Fanuc KAREL source: NC0031.KL

-- PROVISIONAL review KL for V1013-1; original PC SHA256 d6147291fd4dc6949de40ecb1147e79c050cf0ada10eea68c805d8dba57ce3dc
-- Incomplete behavior may be omitted. Consult companion uncertainty JSON. Do not deploy.
PROGRAM NC0031
%NOLOCKGROUP
-- UNRESOLVED_LOCAL_POOL 1 cells at code offset 3; source declarations unknown
-- DIRECT_LOCAL_WORD_ACCESS alone does not prove INTEGER, REAL, or BOOLEAN
BEGIN
  -- UNRESOLVED_PC offsets 0-8; opcodes 2B,2C,7B
  -- UNRESOLVED_PC offsets 13-20; opcodes 9D,23
  -- UNRESOLVED_PC offsets 25-42; opcodes 21,40,41,42
  -- UNRESOLVED_PC offsets 47-64; opcodes 21,40,41,42
  -- UNRESOLVED_PC offsets 69-86; opcodes 21,40,41,42
  -- UNRESOLVED_PC offsets 91-108; opcodes 21,40,41,42
  -- UNRESOLVED_PC offsets 113-130; opcodes 21,40,41,42
  -- UNRESOLVED_PC offsets 135-152; opcodes 21,40,41,42
  -- UNRESOLVED_PC offsets 157-174; opcodes 21,40,41,42
  -- UNRESOLVED_PC offsets 179-196; opcodes 21,40,41,42
  -- UNRESOLVED_PC offsets 201-218; opcodes 21,40,41,42
  -- UNRESOLVED_PC offsets 223-240; opcodes 21,40,41,42
  -- UNRESOLVED_PC offsets 245-262; opcodes 21,40,41,42
  -- UNRESOLVED_PC offsets 267-284; opcodes 21,40,41,42
  -- UNRESOLVED_PC offsets 289-306; opcodes 21,40,41,42
  -- UNRESOLVED_PC offsets 311-328; opcodes 21,40,41,42
  -- UNRESOLVED_PC offsets 333-350; opcodes 21,40,41,42
  -- UNRESOLVED_PC offsets 355-372; opcodes 21,40,41,42
  -- UNRESOLVED_PC offsets 377-394; opcodes 21,40,41,42
  -- UNRESOLVED_PC offsets 399-416; opcodes 21,40,41,42
  -- UNRESOLVED_PC offsets 421-438; opcodes 21,40,41,42
  -- UNRESOLVED_PC offsets 443-460; opcodes 21,40,41,42
  -- UNRESOLVED_PC offsets 465-495; opcodes 21,9D,52,23,7A,40,41,42
  -- UNRESOLVED_PC offsets 500-524; opcodes 21,2E,52,23,7A,43
  -- UNRESOLVED_PC offsets 529-547; opcodes 21,2E,52,23
  -- UNRESOLVED_PC offsets 552-568; opcodes 7A,40,41,42
  -- UNRESOLVED_PC offsets 573-597; opcodes 21,2E,52,23,7A,43
  -- UNRESOLVED_PC offsets 602-620; opcodes 21,2E,52,23
  -- UNRESOLVED_PC offsets 625-641; opcodes 7A,40,41,42
  -- UNRESOLVED_PC offsets 646-670; opcodes 21,2E,52,23,7A,43
  -- UNRESOLVED_PC offsets 675-693; opcodes 21,2E,52,23
  -- UNRESOLVED_PC offsets 698-714; opcodes 7A,40,41,42
  -- UNRESOLVED_PC offsets 719-743; opcodes 21,2E,52,23,7A,43
  -- UNRESOLVED_PC offsets 748-766; opcodes 21,2E,52,23
  -- UNRESOLVED_PC offsets 771-787; opcodes 7A,40,41,42
  -- UNRESOLVED_PC offsets 792-816; opcodes 21,2E,52,23,7A,43
  -- UNRESOLVED_PC offsets 821-839; opcodes 21,2E,52,23
  -- UNRESOLVED_PC offsets 844-860; opcodes 7A,40,41,42
  -- UNRESOLVED_PC offsets 865-889; opcodes 21,2E,52,23,7A,43
  -- UNRESOLVED_PC offsets 894-912; opcodes 21,2E,52,23
  -- UNRESOLVED_PC offsets 917-933; opcodes 7A,40,41,42
  -- UNRESOLVED_PC offsets 938-962; opcodes 21,2E,52,23,7A,43
  -- UNRESOLVED_PC offsets 967-985; opcodes 21,2E,52,23
  -- UNRESOLVED_PC offsets 990-1006; opcodes 7A,40,41,42
  -- UNRESOLVED_PC offsets 1011-1035; opcodes 21,2E,52,23,7A,43
  -- UNRESOLVED_PC offsets 1040-1058; opcodes 21,2E,52,23
  -- UNRESOLVED_PC offsets 1063-1079; opcodes 7A,40,41,42
  -- UNRESOLVED_PC offsets 1084-1108; opcodes 21,2E,52,23,7A,43
  -- UNRESOLVED_PC offsets 1113-1131; opcodes 21,2E,52,23
  -- UNRESOLVED_PC offsets 1136-1152; opcodes 7A,40,41,42
  -- UNRESOLVED_PC offsets 1157-1181; opcodes 21,2E,52,23,7A,43
  -- UNRESOLVED_PC offsets 1186-1204; opcodes 21,2E,52,23
  -- UNRESOLVED_PC offsets 1209-1225; opcodes 7A,40,41,42
  -- UNRESOLVED_PC offsets 1230-1254; opcodes 21,2E,52,23,7A,43
  -- UNRESOLVED_PC offsets 1259-1277; opcodes 21,2E,52,23
  -- UNRESOLVED_PC offsets 1282-1298; opcodes 7A,40,41,42
  -- UNRESOLVED_PC offsets 1303-1327; opcodes 21,2E,52,23,7A,43
  -- UNRESOLVED_PC offsets 1332-1350; opcodes 21,2E,52,23
  -- UNRESOLVED_PC offsets 1355-1371; opcodes 7A,40,41,42
  -- UNRESOLVED_PC offsets 1376-1400; opcodes 21,2E,52,23,7A,43
  -- UNRESOLVED_PC offsets 1405-1423; opcodes 21,2E,52,23
  -- UNRESOLVED_PC offsets 1428-1444; opcodes 7A,40,41,42
  -- UNRESOLVED_PC offsets 1449-1473; opcodes 21,2E,52,23,7A,43
  -- UNRESOLVED_PC offsets 1478-1496; opcodes 21,2E,52,23
  -- UNRESOLVED_PC offsets 1501-1517; opcodes 7A,40,41,42
  -- UNRESOLVED_PC offsets 1522-1546; opcodes 21,2E,52,23,7A,43
  -- UNRESOLVED_PC offsets 1551-1569; opcodes 21,2E,52,23
  -- UNRESOLVED_PC offsets 1574-1590; opcodes 7A,40,41,42
  -- UNRESOLVED_PC offsets 1595-1619; opcodes 21,2E,52,23,7A,43
  -- UNRESOLVED_PC offsets 1624-1642; opcodes 21,2E,52,23
  -- UNRESOLVED_PC offsets 1647-1663; opcodes 7A,40,41,42
  -- UNRESOLVED_PC offsets 1668-1692; opcodes 21,2E,52,23,7A,43
  -- UNRESOLVED_PC offsets 1697-1715; opcodes 21,2E,52,23
  -- UNRESOLVED_PC offsets 1720-1736; opcodes 7A,40,41,42
  -- UNRESOLVED_PC offsets 1741-1765; opcodes 21,2E,52,23,7A,43
  -- UNRESOLVED_PC offsets 1770-1788; opcodes 21,2E,52,23
  -- UNRESOLVED_PC offsets 1793-1809; opcodes 7A,40,41,42
  -- UNRESOLVED_PC offsets 1814-1838; opcodes 21,2E,52,23,7A,43
  -- UNRESOLVED_PC offsets 1843-1861; opcodes 21,2E,52,23
  -- UNRESOLVED_PC offsets 1866-1882; opcodes 7A,40,41,42
  -- UNRESOLVED_PC offsets 1887-1911; opcodes 21,2E,52,23,7A,43
  -- UNRESOLVED_PC offsets 1916-1934; opcodes 21,2E,52,23
  -- UNRESOLVED_PC offsets 1944-1948; opcodes 7F
  -- UNRESOLVED_PC offsets 1953-1957; opcodes 27,AA
  -- UNRESOLVED_PC offsets 1962-1966; opcodes 7F
END NC0031
